# EPICS substitutions: vme_iocs/iocbio4/iocBoot/asynRecord.substitutions
file "$(ASYN)/db/asynRecord.db"
{
pattern
{P        R         PORT    ADDR    OMAX  IMAX}
{18ID:     asyn_1   serial1    0     256  256}
{18ID:     asyn_2   serial2    0     256  256}
{18ID:     asyn_3   serial3    0     256  256}
{18ID:     asyn_4   serial4    0     256  256}
{18ID:     asyn_5   serial5    0     256  256}
{18ID:     asyn_6   serial6    0    2600  2600}
{18ID:     asyn_7   serial7    0     256  256}
{18ID:     asyn_8   serial8    0     256  256}
{18ID:     gpib1    gpib1      1    2600 2600}
}
